(* Schneider Machine Expert - Basic project M221-KSB-single-pump, file version 1.8.0.0 *)
(* ProjectInformations: Name=New project *)

HARDWARE
  Cpu 0: TM221CE24R
  ModuleExtensionObject 0: TM3TI4/G
  ModuleExtensionObject 1: TM3TI8T/G
  ModuleExtensionObject 2: TM3AI2H/G
  EthernetConfiguration: NetworkName=M221, IpAllocationMode=FixedAddress, IpAddress=0.0.0.0, SubnetMask=0.0.0.0
  SerialLineConfiguration: Baud=Baud19200, Parity=ParityEven, DataBits=DataBits8, StopBits=StopBits1, PhysicalMedium=PhysicalMediumRs485, TransmissionMode=TransmissionModeModbusRtu, SlaveId=1, Addressing=SlaveAddressing
  MastTask: UsePeriodScanMode=false, PeriodScan=100
  FastTask: Period=255
  CpuBehavior: StartingMode=StartAsPreviousState, AutoSaveRamOnEeprom=true, WatchdogPeriod=250

SYMBOLS  (address, symbol, comment, settings)
  %M0       WINDING_TEMP_ALARM
  %M1       SEAL_FAIL_ALARM
  %M2       HIGH_FLOAT_ALARM
  %M3       VIBRATION_ALARM
  %M4       HIGH_RTD_ALARM
  %M5       RESET_ALARMS
  %M6       SILENCE_ALARMS
  %M7       WINDING_TEMP_ALARM_BYPASS
  %M8       SEAL_FAIL_ALARM_BYPASS
  %M9       HIGH_FLOAT_ALARM_BYPASS
  %M10      VIBRATION_ALARM_BYPASS
  %M11      HIGH_RTD_ALARM_BYPASS
  %MW0      WINDING1_TEMP_SETPOINT
  %MW1      WINDING2_TEMP_SETPOINT
  %MW2      WINDING3_TEMP_SETPOINT
  %MW3      BOTTOM_BEARING_SETPOINT
  %MW4      VIBRATION_SETPOINT
  %KW0      DISCONNECTED_VALUE  [Value=-32768]
  %TM0      HIGH_BOT_BEARING_TMP_ALARM_DELAY
  %TM1      HIGH_FLOAT_ALARM_DELAY
  %TM2      HIGH_WINDING_TEMP_ALARM_DELAY
  %TM3      SEAL_FAIL_ALARM_DELAY
  %TM4      VIBRATION_ALARM_DELAY
  %I0.0     SEAL_FAIL  "Reversed Logic Sensor!!! Normally Closed. Seal failing breaks connection"
  %I0.1     HIGH_FLOAT
  %Q0.0     PUMP_ENABLE
  %Q0.1     AUDIBLE_ALARM
  %IW1.0    WINDING1_TEMP  [Type=Type_PT100, Scope=Scope_Customized, Minimum=-32768, Maximum=32767]
  %IW1.1    WINDING2_TEMP  [Type=Type_PT100, Scope=Scope_Customized, Minimum=-32768, Maximum=32767]
  %IW1.2    WINDING3_TEMP  [Type=Type_PT100, Scope=Scope_Customized, Minimum=-32768, Maximum=32767]
  %IW1.3    BOTTOM_BEARING_TEMP  [Type=Type_PT100, Scope=Scope_Customized, Minimum=-32768, Maximum=32767]
  %IW2.0    WINDING_TEMP  [Type=Type_PTC, Scope=Scope_Threshold, Minimum=100, Maximum=10000]
  %IW3.0    VIBRATION  [Type=Type_4_20mA, Scope=Scope_Customized, Minimum=4000, Maximum=20000]

POU Alarm Calculations
  (* SectionNumber=0 *)

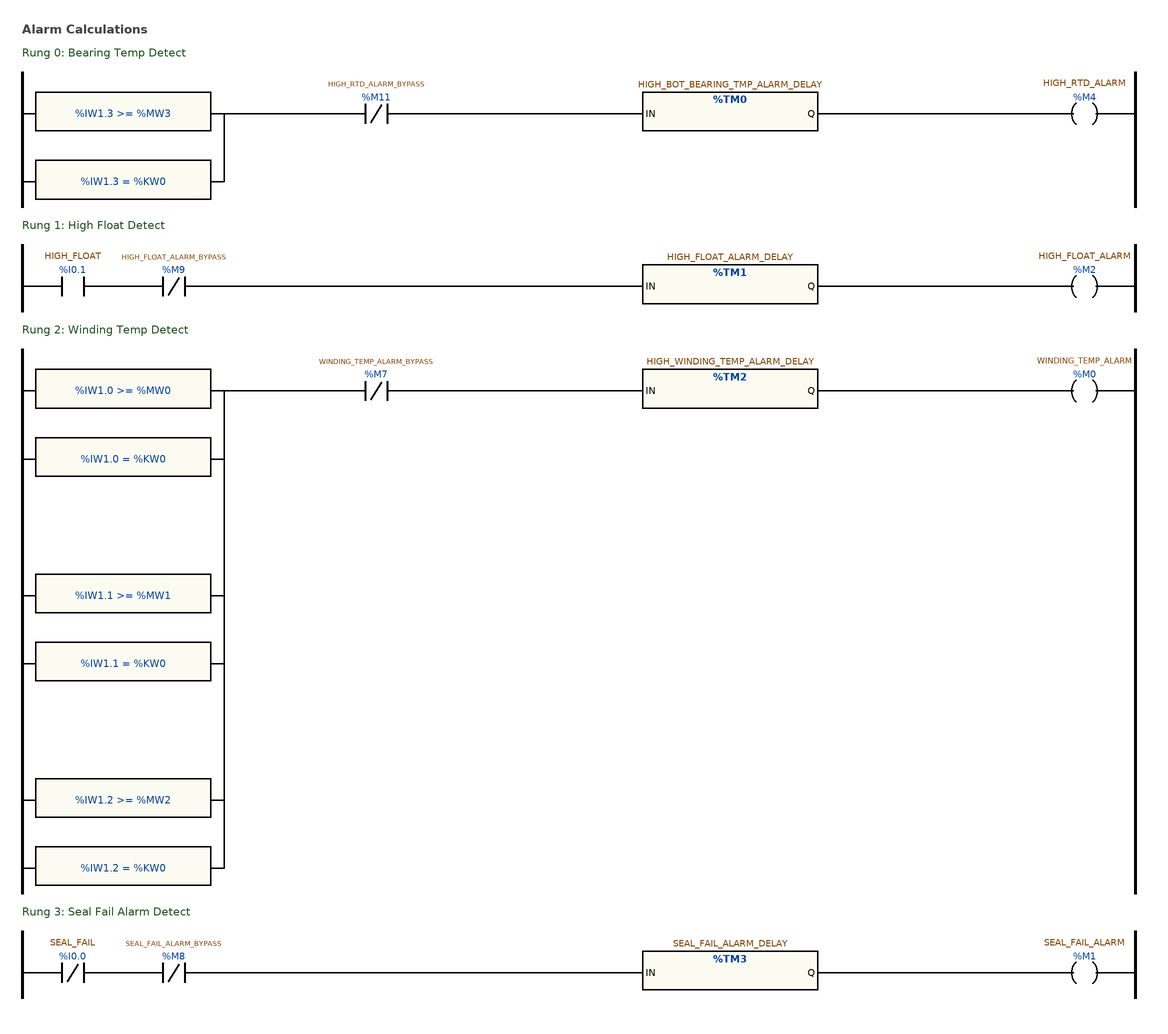

// Rung 0: Bearing Temp Detect
  BLK %TM0                (* HIGH_BOT_BEARING_TMP_ALARM_DELAY *)
  LD [ %IW1.3 >= %MW3 ]   (* BOTTOM_BEARING_TEMP, BOTTOM_BEARING_SETPOINT *)
  OR [ %IW1.3 = %KW0 ]    (* BOTTOM_BEARING_TEMP, DISCONNECTED_VALUE *)
  ANDN %M11               (* HIGH_RTD_ALARM_BYPASS *)
  IN
  OUT_BLK
  LD Q
  ST %M4                  (* HIGH_RTD_ALARM *)
  END_BLK
  // as ST:
  //   HIGH_BOT_BEARING_TMP_ALARM_DELAY(IN := (BOTTOM_BEARING_TEMP >= BOTTOM_BEARING_SETPOINT OR BOTTOM_BEARING_TEMP = DISCONNECTED_VALUE) AND NOT HIGH_RTD_ALARM_BYPASS);
  //   HIGH_RTD_ALARM := HIGH_BOT_BEARING_TMP_ALARM_DELAY.Q;

// Rung 1: High Float Detect
  BLK %TM1                (* HIGH_FLOAT_ALARM_DELAY *)
  LD %I0.1                (* HIGH_FLOAT *)
  ANDN %M9                (* HIGH_FLOAT_ALARM_BYPASS *)
  IN
  OUT_BLK
  LD Q
  ST %M2                  (* HIGH_FLOAT_ALARM *)
  END_BLK
  // as ST:
  //   HIGH_FLOAT_ALARM_DELAY(IN := HIGH_FLOAT AND NOT HIGH_FLOAT_ALARM_BYPASS);
  //   HIGH_FLOAT_ALARM := HIGH_FLOAT_ALARM_DELAY.Q;

// Rung 2: Winding Temp Detect
  BLK %TM2                (* HIGH_WINDING_TEMP_ALARM_DELAY *)
  LD [ %IW1.0 >= %MW0 ]   (* WINDING1_TEMP, WINDING1_TEMP_SETPOINT *)
  OR [ %IW1.0 = %KW0 ]    (* WINDING1_TEMP, DISCONNECTED_VALUE *)
  OR [ %IW1.1 >= %MW1 ]   (* WINDING2_TEMP, WINDING2_TEMP_SETPOINT *)
  OR [ %IW1.1 = %KW0 ]    (* WINDING2_TEMP, DISCONNECTED_VALUE *)
  OR [ %IW1.2 >= %MW2 ]   (* WINDING3_TEMP, WINDING3_TEMP_SETPOINT *)
  OR [ %IW1.2 = %KW0 ]    (* WINDING3_TEMP, DISCONNECTED_VALUE *)
  ANDN %M7                (* WINDING_TEMP_ALARM_BYPASS *)
  IN
  OUT_BLK
  LD Q
  ST %M0                  (* WINDING_TEMP_ALARM *)
  END_BLK
  // as ST:
  //   HIGH_WINDING_TEMP_ALARM_DELAY(IN := (WINDING1_TEMP >= WINDING1_TEMP_SETPOINT OR WINDING1_TEMP = DISCONNECTED_VALUE OR WINDING2_TEMP >= WINDING2_TEMP_SETPOINT OR WINDING2_TEMP = DISCONNECTED_VALUE OR WINDING3_TEMP >= WINDING3_TEMP_SETPOINT OR WINDING3_TEMP = DISCONNECTED_VALUE) AND NOT WINDING_TEMP_ALARM_BYPASS);
  //   WINDING_TEMP_ALARM := HIGH_WINDING_TEMP_ALARM_DELAY.Q;

// Rung 3: Seal Fail Alarm Detect
  BLK %TM3                (* SEAL_FAIL_ALARM_DELAY *)
  LDN %I0.0               (* SEAL_FAIL *)
  ANDN %M8                (* SEAL_FAIL_ALARM_BYPASS *)
  IN
  OUT_BLK
  LD Q
  ST %M1                  (* SEAL_FAIL_ALARM *)
  END_BLK
  // as ST:
  //   SEAL_FAIL_ALARM_DELAY(IN := NOT SEAL_FAIL AND NOT SEAL_FAIL_ALARM_BYPASS);
  //   SEAL_FAIL_ALARM := SEAL_FAIL_ALARM_DELAY.Q;

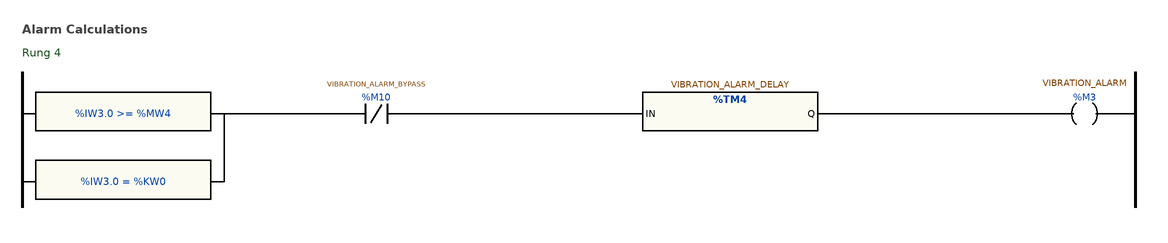

// Rung 4
  BLK %TM4                (* VIBRATION_ALARM_DELAY *)
  LD [ %IW3.0 >= %MW4 ]   (* VIBRATION, VIBRATION_SETPOINT *)
  OR [ %IW3.0 = %KW0 ]    (* VIBRATION, DISCONNECTED_VALUE *)
  ANDN %M10               (* VIBRATION_ALARM_BYPASS *)
  IN
  OUT_BLK
  LD Q
  ST %M3                  (* VIBRATION_ALARM *)
  END_BLK
  // as ST:
  //   VIBRATION_ALARM_DELAY(IN := (VIBRATION >= VIBRATION_SETPOINT OR VIBRATION = DISCONNECTED_VALUE) AND NOT VIBRATION_ALARM_BYPASS);
  //   VIBRATION_ALARM := VIBRATION_ALARM_DELAY.Q;
